// TIA Portal V20 export
DATA_BLOCK "InstComRF160B"   // DB281
TITLE = InstComRF160B
VERSION : 1.0
// stored: InstanceOfName ComRF160B, InstanceOfType FB
"ComRF160B"
   // VAR_INPUT
   //    enable { ExternalAccessible := 'False'; ExternalVisible := 'False'; ExternalWritable := 'False'} : Bool;
   //    cont { ExternalAccessible := 'False'; ExternalVisible := 'False'; ExternalWritable := 'False'} : Bool;
   //    localPort { ExternalAccessible := 'False'; ExternalVisible := 'False'; ExternalWritable := 'False'} : UInt;
   //    interfaceId { ExternalAccessible := 'False'; ExternalVisible := 'False'; ExternalWritable := 'False'} : HW_ANY;
   //    connectionId { ExternalAccessible := 'False'; ExternalVisible := 'False'; ExternalWritable := 'False'} : CONN_OUC;
   // END_VAR
   // VAR_OUTPUT
   //    error { ExternalAccessible := 'False'; ExternalVisible := 'False'; ExternalWritable := 'False'} : Bool;
   //    done { ExternalAccessible := 'False'; ExternalVisible := 'False'; ExternalWritable := 'False'} : Bool;
   //    connected { ExternalAccessible := 'False'; ExternalVisible := 'False'; ExternalWritable := 'False'} : Bool;
   //    restart { ExternalAccessible := 'False'; ExternalVisible := 'False'; ExternalWritable := 'False'} : Bool;
   //    lenEpcId { ExternalAccessible := 'False'; ExternalVisible := 'False'; ExternalWritable := 'False'} : Byte;
   //    lenData { ExternalAccessible := 'False'; ExternalVisible := 'False'; ExternalWritable := 'False'} : Byte;
   //    status { ExternalAccessible := 'False'; ExternalVisible := 'False'; ExternalWritable := 'False'} : Word;
   //    statusId { ExternalAccessible := 'False'; ExternalVisible := 'False'; ExternalWritable := 'False'} : UInt;
   // END_VAR
   // VAR_IN_OUT
   //    reset { ExternalAccessible := 'False'; ExternalVisible := 'False'; ExternalWritable := 'False'} : Bool;
   //    data : Variant;
   //    epcId : Variant;
   // END_VAR
   // VAR
   //    statConnectionData { ExternalAccessible := 'False'; ExternalVisible := 'False'; ExternalWritable := 'False'; S7_SetPoint := 'True'} : TCON_IP_v4;
   //    instTRCV { ExternalAccessible := 'False'; ExternalVisible := 'False'; ExternalWritable := 'False'; S7_SetPoint := 'True'} : TRCV_C;
   //    statRCV { ExternalAccessible := 'False'; ExternalVisible := 'False'; ExternalWritable := 'False'} : Struct
   //       Enable : Bool;
   //       Cont : Bool;
   //       Len : UDInt;
   //       Done : Bool;
   //       Busy : Bool;
   //       Error : Bool;
   //       Status : Word;
   //       RcvLen : UDInt;
   //       DataValues : Array[0..311] of Byte;
   //       COM_RST : Bool;
   //       ADDR : Bool;
   //    END_STRUCT;
   //    statErrorRcv { ExternalAccessible := 'False'; ExternalVisible := 'False'; ExternalWritable := 'False'} : Bool;
   //    statLastErrorStatus { ExternalAccessible := 'False'; ExternalVisible := 'False'; ExternalWritable := 'False'} : Word;
   //    statBufferPtr { ExternalAccessible := 'False'; ExternalVisible := 'False'; ExternalWritable := 'False'} : UDInt;
   //    statRCVBufferValues { ExternalAccessible := 'False'; ExternalVisible := 'False'; ExternalWritable := 'False'} : Array[0..1000] of Byte;
   // END_VAR
BEGIN
END_DATA_BLOCK
